// Mitsubishi GX Works2 project: 11   PLC: FX3U/FX3UC

PROGRAM MAIN
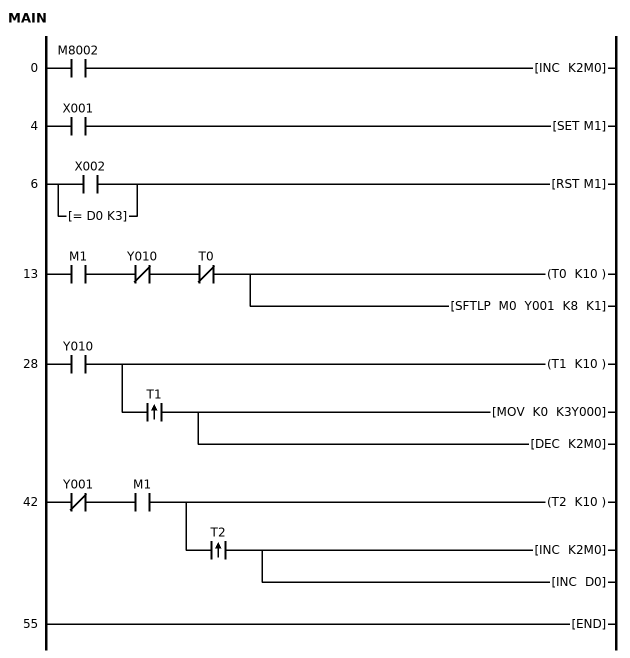
0     LD      M8002
      INC     K2M0
4     LD      X001
      SET     M1
6     LD      X002
      OR=     D0 K3
      RST     M1
13    LD      M1
      ANI     Y010
      ANI     T0
      OUT     T0 K10
      SFTLP   M0 Y001 K8 K1
28    LD      Y010
      OUT     T1 K10
      ANDP    T1
      MOV     K0 K3Y000
      DEC     K2M0
42    LDI     Y001
      AND     M1
      OUT     T2 K10
      ANDP    T2
      INC     K2M0
      INC     D0
55    END
END_PROGRAM
